PROGRAM MAIN
VAR
	dt1:DT;
	r1:REAL;
	r2:LREAL;
	i1:INT;
	i2:UDINT;
END_VAR

prgTrigTesting();

END_PROGRAM

(* stored: Version 1.1.0.1, ProductVersion 3.1.4024.11
   POU MAIN: Id {077b38a9-d9d0-4582-9d08-e7ea990f2571}, SpecialFunc None *)
